{attribute addProperty BoxType "EK1100-0000-0018"}
{attribute addProperty Id "Beckhoff_EPP9xxxEK1122Beckhoff_EPP9xxxEK1122_703EDA8E56070"}
{attribute addProperty CRC "1803377247"}
{attribute addProperty SizeInBites "560"}
{attribute addProperty SizeInBytes "70"}
TYPE Beckhoff_EPP9xxx_6B7D5A5F EXTENDS EK1100_179A0949 :
STRUCT
	{attribute addProperty Name "Beckhoff_EPP9xxxEK1122"}
	Beckhoff_EPP9xxxEK1122 : Beckhoff_EPP9xxxEK1122_703EDA8E;
END_STRUCT
END_TYPE

(* stored: Version 1.2.0.0, ProductVersion 3.1.4024.9
   DUT Beckhoff_EPP9xxx_6B7D5A5F: Id {f23e1522-3fee-49b3-bc1b-c60e2199f582} *)
